// TwinCAT 3 PLC project Example
// ProgramVersion: 3.1.4022.7
// libraries:
//   lcls-twincat-motion, * (SLAC)
//   Tc2_Standard, * (Beckhoff Automation GmbH)
//   Tc2_System, * (Beckhoff Automation GmbH)
//   Tc2_Utilities, * (Beckhoff Automation GmbH)
//   Tc3_Module, * (Beckhoff Automation GmbH)
// project tree:
//   / PlcTask.TcTTO (not stored)
//   POUs/ Main.TcPOU

// ---- POUs/Main.TcPOU
PROGRAM Main
VAR
    // Simulated motor that is always allowed to move
    {attribute 'pytmc' := '
        pv: PLC:TST:MOT:SIM:01
        field: DESC Simulated Working Motor
    '}
    M1: DUT_MotionStage;
    fbMotion1: FB_MotionStageSim;

    // Simulated motor that is never allowed to move
    {attribute 'pytmc' := '
        pv: PLC:TST:MOT:SIM:02
        field: DESC Simulated Broken Motor
    '}
    M2: DUT_MotionStage;
    fbMotion2: FB_MotionStage;

    // Simulated motor with limits at 0 and 100
    {attribute 'pytmc' := '
        pv: PLC:TST:MOT:SIM:03
        field: DESC Simulated Working Motor With Limits
    '}
    M3: DUT_MotionStage;
    fbMotion3: FB_MotionStage;
    
    {attribute 'pytmc' := '
        pv: PLC:TST:MOT:TC:RESTART
        field: DESC Set to True to restart TwinCAT
        field: ZRST False
        field: ONST True
    '}
    bTCRestart: BOOL;
    fbTCRestart: TC_Restart;
END_VAR

fbMotion1(stMotionStage := M1);
fbMotion2(stMotionStage := M2);
fbMotion3(stMotionStage := M3);
M3.bHardwareEnable := TRUE;
M3.bPowerSelf := TRUE;
M3.bLimitForwardEnable := M3.Axis.NcToPlc.ActPos < 99.7;
M3.bLimitBackwardEnable := M3.Axis.NcToPlc.ActPos > 0.2;

fbTCRestart(
    NETID := '',
    RESTART := bTCRestart);

END_PROGRAM
